// TwinCAT 3 PLC project PLC1
// ProgramVersion: 3.1.4026.18
// libraries:
//   Tc2_MC2, * (Beckhoff Automation GmbH)
//   Tc2_Standard, * (Beckhoff Automation GmbH)
//   Tc2_System, * (Beckhoff Automation GmbH)
// project tree:
//   / ClassDiagram.TcCD (not stored), PlcTask.TcTTO
//   GVLs/ GVL.TcGVL, SETTINGS.TcGVL
//   POUs/ Galaxy.TcPOU, MAIN.TcPOU
//   _MoverLink/Base/ Base.TcPOU, I_Base.TcIO (not stored)
//   _MoverLink/Manager/ I_RegisterMover.TcIO (not stored), I_RegisterPosition.TcIO, Manager.TcPOU
//   _MoverLink/Mode/ E_Mode.TcDUT (not stored), I_Mode.TcIO (not stored), Mode.TcPOU
//   _MoverLink/Mover/ I_Mover.TcIO, I_MoverPos.TcIO (not stored), Mover.TcPOU (not stored)
//   _MoverLink/Position/ I_Position.TcIO, I_PosMover.TcIO, I_PosStation.TcIO, Position.TcPOU
//   _MoverLink/Station/ I_Station.TcIO, Station.TcPOU (not stored)
//   _MoverLink/User/ User.TcPOU (not stored)
// real-time tasks:
//   TASK PlcTask: cycle T#10ms, priority 20, ADS port 350

CONFIGURATION PLC1
    RESOURCE PLC ON TwinCAT3
        TASK PlcTask(INTERVAL := T#10ms, PRIORITY := 20);
        PROGRAM MAIN WITH PlcTask : MAIN;
    END_RESOURCE
END_CONFIGURATION

// ---- GVLs/GVL.TcGVL
{attribute 'qualified_only'}
VAR_GLOBAL
	monitorValue : UDINT;
	monitorReal	: LREAL;
END_VAR

// ---- GVLs/SETTINGS.TcGVL
{attribute 'qualified_only'}
VAR_GLOBAL CONSTANT
	MAX_MOVERS			: INT 	:= 10;
	MAX_POSITIONS		: INT 	:= 10;
	MAX_POS_STATIONS	: INT 	:= 5;
	MAX_DEVICES 		: UDINT	:= 30;
	TRACK_LENGTH 		: LREAL := 3000;
END_VAR

// ---- _MoverLink/Manager/I_RegisterPosition.TcIO
INTERFACE I_RegisterPosition

METHOD RegisterPosition : BOOL
VAR_INPUT
	position : I_Position;
END_VAR
END_METHOD

END_INTERFACE

// ---- _MoverLink/Mover/I_Mover.TcIO
INTERFACE I_Mover EXTENDS I_MoverPos

METHOD Cyclic : BOOL
VAR_INPUT
END_VAR
END_METHOD

PROPERTY ErrorCode : UDINT
GET
END_GET
END_PROPERTY

PROPERTY Linked : BOOL
GET
END_GET
END_PROPERTY

METHOD SetPosLink : BOOL
VAR_INPUT
	position : I_PosMover;
END_VAR
END_METHOD

PROPERTY State : UDINT
GET
END_GET
SET
END_SET
END_PROPERTY

PROPERTY Step : UDINT
GET
END_GET
END_PROPERTY

METHOD Unlink : BOOL
VAR_INPUT
END_VAR
END_METHOD

METHOD Update : BOOL
VAR_INPUT
END_VAR
END_METHOD

END_INTERFACE

// ---- _MoverLink/Position/I_Position.TcIO
INTERFACE I_Position EXTENDS I_PosMover

PROPERTY RequestedStep : INT
GET
END_GET
SET
END_SET
END_PROPERTY

PROPERTY RequestMover : BOOL
GET
END_GET
END_PROPERTY

METHOD SetMoverLink : BOOL
VAR_INPUT
	mover : I_MoverPos;
END_VAR
END_METHOD

END_INTERFACE

// ---- _MoverLink/Position/I_PosMover.TcIO
INTERFACE I_PosMover

PROPERTY TargetPosition : LREAL
GET
END_GET
END_PROPERTY

END_INTERFACE

// ---- _MoverLink/Position/I_PosStation.TcIO
INTERFACE I_PosStation

METHOD EnableRequest : BOOL
VAR_INPUT
	OnOff : BOOL;
END_VAR
END_METHOD

PROPERTY InPosition : BOOL
GET
END_GET
END_PROPERTY

PROPERTY Linked : BOOL
GET
END_GET
END_PROPERTY

METHOD MoverChangeStep : BOOL
VAR_INPUT
	step : UDINT;
END_VAR
END_METHOD

PROPERTY RequestedStep : INT
SET
END_SET
END_PROPERTY

METHOD SetAttractStep : BOOL
VAR_INPUT
	step : INT;
END_VAR
END_METHOD

END_INTERFACE

// ---- _MoverLink/Station/I_Station.TcIO
INTERFACE I_Station

METHOD Clear : BOOL
VAR_INPUT
END_VAR
END_METHOD

METHOD Enable : BOOL
VAR_INPUT
END_VAR
END_METHOD

PROPERTY InPosition : BOOL
GET
END_GET
END_PROPERTY

METHOD JobDone : BOOL
VAR_INPUT
END_VAR
END_METHOD

METHOD SetPosAttractStep : BOOL
VAR_INPUT
	step : INT;
END_VAR
END_METHOD

METHOD SetPosMoverStep : BOOL
VAR_INPUT
	posIndex	: INT;
	step		: INT;
END_VAR
END_METHOD

END_INTERFACE

// ---- POUs/MAIN.TcPOU
PROGRAM MAIN
VAR
	Galaxy : Galaxy;
END_VAR

// Init - First Scan Done before run Galaxy
IF NOT Galaxy.IsInitialized THEN
	Galaxy.Init();
	RETURN;
END_IF

// Cyclic
Galaxy();

END_PROGRAM

// ---- POUs/Galaxy.TcPOU
FUNCTION_BLOCK Galaxy
VAR
	Manager 	: Manager;
	Mode		: Mode;
	Mover_01 	: Mover(ID := 101, mode := Mode, manager := Manager);
	Mover_02 	: Mover(ID := 102, mode := Mode, manager := Manager);
	Station_A 	: Station;
	Position_11 : Position(position := 1000, manager := Manager);
	Position_12 : Position(position := 0900, manager := Manager);
	Station_B 	: Station;
	Position_21 : Position(position := 1500, manager := Manager);
	Position_22 : Position(position := 1400, manager := Manager);
	User		: User(Station_A, Station_B);
	
	// Flags
	_initialized	: BOOL;
	_configDone 	: BOOL;
	
	dummy 			: BOOL;
END_VAR

// Config
IF NOT _configDone THEN
	Station_A.RegisterPosition(Position_11);
	Station_A.RegisterPosition(Position_12);	
	Station_B.RegisterPosition(Position_21);
	Station_B.RegisterPosition(Position_22);
	_configDone := TRUE;		
END_IF

// User Interfaces
User();

// Cycle
Station_A.Cyclic();
Station_B.Cyclic();
Manager.Cyclic();

METHOD Init : BOOL
VAR_INPUT
END_VAR
// Logic

_initialized := TRUE;
END_METHOD

PROPERTY IsInitialized : BOOL
GET
IsInitialized := _initialized;
END_GET
END_PROPERTY

END_FUNCTION_BLOCK

// ---- _MoverLink/Manager/Manager.TcPOU
FUNCTION_BLOCK Manager IMPLEMENTS I_RegisterMover, I_RegisterPosition
VAR CONSTANT
	MAX_MOVERS 		: INT := 10;
	MAX_POSITIONS	: INT := 10;
END_VAR
VAR
	_IMover 		: ARRAY [1..SETTINGS.MAX_MOVERS] OF I_Mover;
	_moverCount 	: INT;
	_IPos	: ARRAY [1..SETTINGS.MAX_POSITIONS] OF I_Position;
	_PosCount : INT;
END_VAR

METHOD PRIVATE _FindUnlinkedMoverWithStep : I_Mover
VAR_INPUT
	MoverStep : UDINT;
END_VAR
VAR
	i : INT;
END_VAR
FOR i:=1 TO _moverCount DO
	IF _IMover[i].Step = MoverStep AND NOT _IMover[i].Linked THEN
		_FindUnlinkedMoverWithStep := _IMover[i];	
	END_IF
END_FOR
END_METHOD

METHOD Cyclic : BOOL
VAR_INPUT
END_VAR
VAR
	i : INT;
	StepRequest : UDINT;
	IMover		: I_Mover;
	IMoverPos 	: I_MoverPos;
END_VAR
// Call Positions
IMover := 0;
FOR i:=1 TO _PosCount DO
	IF _IPos[i].RequestMover THEN
		IMover := _FindUnlinkedMoverWithStep(_Ipos[i].RequestedStep);
		IF IMover <> 0 THEN
			_Ipos[i].SetMoverLink(IMover);
			IMover.SetPosLink(_IPos[i]);	
		END_IF	
	END_IF
END_FOR

// Call Movers
FOR i:=1 TO _moverCount DO
	_IMover[i].Cyclic();
END_FOR
END_METHOD

METHOD RegisterMover : BOOL
VAR_INPUT
	mover : I_Mover;
END_VAR
VAR
	i : INT;
END_VAR
IF _moverCount < SETTINGS.MAX_MOVERS THEN
//	IF mover <> 0 THEN
		_moverCount := _moverCount + 1;
		_IMover[_moverCount] := mover;
		RegisterMover := TRUE;	
//	END_IF
END_IF
END_METHOD

METHOD RegisterPosition : BOOL
VAR_INPUT
	position : I_Position;
END_VAR
VAR
	i : INT;
END_VAR
IF _PosCount < SETTINGS.MAX_POSITIONS THEN
	IF position <> 0 THEN
		_PosCount := _PosCount + 1;
		_IPos[_PosCount] := position;
		RegisterPosition := TRUE;	
	END_IF
END_IF
END_METHOD

END_FUNCTION_BLOCK

// ---- _MoverLink/Position/Position.TcPOU
FUNCTION_BLOCK Position IMPLEMENTS I_Position, I_PosStation
VAR_INPUT
END_VAR
VAR_OUTPUT
END_VAR
VAR
	_position		: LREAL;
	_enableRequest 	: BOOL;
	_IMover			: I_MoverPos;
	_requestStep 	: INT;
	_posID				: UDINT;
END_VAR

METHOD EnableRequest : BOOL
VAR_INPUT
	OnOff : BOOL;
END_VAR
_EnableRequest := OnOff;
EnableRequest := RequestMover;
END_METHOD

//FB_Init is always available implicitly and it is used primarily for initialization.
//The return value is not evaluated. For a specific influence, you can also declare the
//methods explicitly and provide additional code there with the standard initialization
//code. You can evaluate the return value.
METHOD FB_Init: BOOL
VAR_INPUT
    bInitRetains: BOOL; // TRUE: the retain variables are initialized (reset warm / reset cold)
    bInCopyCode: BOOL;  // TRUE: the instance will be copied to the copy code afterward (online change)
	position : LREAL;  
	manager : I_RegisterPosition; 
END_VAR
_position := position;
manager.RegisterPosition(THIS^);
END_METHOD

{warning 'Add property implementation'}
PROPERTY InPosition : BOOL
GET
VAR
	difference	: LREAL;
	tolerance 	: LREAL := 100;
END_VAR
IF _IMover <> 0 THEN
	difference := ABS(_position - _IMover.Position);
	IF difference < tolerance THEN
		InPosition := TRUE;
	END_IF	
END_IF
END_GET
END_PROPERTY

PROPERTY Linked : BOOL
GET
Linked := _IMover <> 0;
END_GET
END_PROPERTY

METHOD MoverChangeStep : BOOL
VAR_INPUT
	step	: UDINT;
END_VAR
IF _IMover <> 0 THEN
	_IMover.ChangeStep(step);
END_IF
END_METHOD

PROPERTY RequestedStep : INT
GET
RequestedStep := _requestStep;
END_GET
SET
_requestStep := RequestedStep;
END_SET
END_PROPERTY

{warning 'Add property implementation'}
PROPERTY RequestMover : BOOL
GET
IF _IMover <> 0 THEN
	_enableRequest := FALSE;
END_IF
RequestMover := _enableRequest;
END_GET
END_PROPERTY

METHOD SetAttractStep : BOOL
VAR_INPUT
	step	: INT;
END_VAR
_requestStep := step;
END_METHOD

METHOD SetMoverLink : BOOL
VAR_INPUT
	mover : I_MoverPos;
END_VAR
_IMover := mover;
END_METHOD

PROPERTY TargetPosition : LREAL
GET
TargetPosition := _position;
END_GET
END_PROPERTY

END_FUNCTION_BLOCK

// ---- _MoverLink/Mode/Mode.TcPOU
FUNCTION_BLOCK Mode IMPLEMENTS I_Mode
VAR_INPUT
END_VAR
VAR_OUTPUT
END_VAR
VAR
	_mode : E_Mode;
END_VAR

PROPERTY Mode : E_Mode
GET
Mode := _mode;
END_GET
END_PROPERTY

END_FUNCTION_BLOCK

// ---- _MoverLink/Base/Base.TcPOU
FUNCTION_BLOCK Base
VAR_INPUT
END_VAR
VAR_OUTPUT
END_VAR
VAR
END_VAR

END_FUNCTION_BLOCK
